(* IEC 61131-3 sources: com.logicals.lc3.webinar/logicals_Lib_Webinar/logicals_Webinar_Basic_Lib/logicals_Lib/src_FB_FBD/Logic, 6 files *)

(* ---- FB_lc_EinsAusDrei_Auswahl2_FBD.iecfbd ---- *)
NAMESPACE com.logicals.Basic.Logic
FUNCTION_BLOCK FB_lc_EinsAusDrei_Auswahl2_FBD
  {
    height := 50;
    width := 370;
  }

  VAR_INPUT
    vix_In1 : BOOL;
    vix_In2 : BOOL;
    vix_In3 : BOOL;
  END_VAR
  VAR_OUTPUT
    vox_Out : BOOL;
  END_VAR

  (*

    // Network 1:
    AND(IN1 := vix_In1, IN2 := NOT vix_In2, IN3 := NOT vix_In3, AND => @C(13).AND);
    AND(IN1 := NOT vix_In1, IN2 := vix_In2, IN3 := NOT vix_In3, AND => @C(14).AND);
    AND(IN1 := NOT vix_In1, IN2 := NOT vix_In2, IN3 := vix_In3, AND => @C(16).AND);
    OR(IN1 := @C(13).AND, IN2 := @C(14).AND, IN3 := @C(16).AND, OR => vox_Out);

  *)

  @VF(1) : @E(vix_In1), @R(560.0, 210.0, 140.0, 19.0);
  @VF(2) : @E(vix_In2), @R(560.0, 230.0, 140.0, 19.0);
  @VF(3) : @E(vix_In3), @R(560.0, 250.0, 140.0, 19.0);
  @VF(8) : @E(vox_Out), @R(1200.0, 210.0, 140.0, 19.0);
  @CF(11) : @R(30.0, 40.0, 870.0, 100.0), @T("E:$NFB_lc_EinsAusDreiAuswahl2_FBD"), @POU;
  @CF(12) : @R(1008.0, 42.6, 870.0, 100.0), @T("D:$NFB_lc_EinsAusDreiAuswahl2_FBD"), @POU;
  @C(13) : @F(AND), @R(880.0, 210.0, 40.0, 58.0), BOOL, @I(@N(IN1), @L(9.5)), @I(@N(IN2), @L(29.5), @NEG), @I(@N(IN3), @L(49.5), @NEG), @O(@N(AND), @R(9.5));
  @C(14) : @F(AND), @R(880.0, 310.0, 40.0, 58.0), BOOL, @I(@N(IN1), @L(9.5), @NEG), @I(@N(IN2), @L(29.5)), @I(@N(IN3), @L(49.5), @NEG), @O(@N(AND), @R(9.5));
  @C(15) : @F(OR), @R(1090.0, 210.0, 40.0, 58.0), BOOL, @I(@N(IN1), @L(9.5)), @I(@N(IN2), @L(29.5)), @I(@N(IN3), @L(49.5)), @O(@N(OR), @R(9.5));
  @C(16) : @F(AND), @R(880.0, 410.0, 40.0, 58.0), BOOL, @I(@N(IN1), @L(9.5), @NEG), @I(@N(IN2), @L(29.5), @NEG), @I(@N(IN3), @L(49.5)), @O(@N(AND), @R(9.5));
  @CP(4) : 731.9, 219.5;
  @CP(5) : 731.9, 317.9;
  @CP(6) : 761.0, 239.5;
  @CP(7) : 761.0, 338.2;
  @CP(9) : 790.2, 259.5;
  @CP(10) : 790.2, 354.7;

  @G(17) :
     @L(@VF(1).o, @CP(4)),
     @L(@CP(4), @C(13).IN1),
     @L(@CP(4), @CP(5)),
     @L(@CP(5), @C(14).IN1),
     @L(@CP(5), @C(16).IN1)
    ;
  @G(18) :
     @L(@VF(2).o, @CP(6)),
     @L(@CP(6), @C(13).IN2),
     @L(@CP(6), @CP(7)),
     @L(@CP(7), @C(14).IN2),
     @L(@CP(7), @C(16).IN2)
    ;
  @G(19) :
     @L(@VF(3).o, @CP(9)),
     @L(@CP(9), @C(13).IN3),
     @L(@CP(9), @CP(10)),
     @L(@CP(10), @C(14).IN3),
     @L(@CP(10), @C(16).IN3)
    ;
  @G(23) :
     @L(@C(13).AND, @C(15).IN1)
    ;
  @G(24) :
     @L(@C(14).AND, @C(15).IN2)
    ;
  @G(25) :
     @L(@C(15).OR, @VF(8).i)
    ;
  @G(27) :
     @L(@C(16).AND, @C(15).IN3)
    ;
END_FUNCTION_BLOCK
END_NAMESPACE

(* ---- FB_lc_EinsAusDrei_Auswahl3_FBD.iecfbd ---- *)
NAMESPACE com.logicals.Basic.Logic
FUNCTION_BLOCK FB_lc_EinsAusDrei_Auswahl3_FBD
  {
    width := 350;
    minWidth := 340;
    maxWidth := 340;
    height := 58;
    minHeight := 58;
    maxHeight := 58;
  }

  VAR_INPUT
    vix_In1 : BOOL;
    vix_In2 : BOOL;
    vix_In3 : BOOL;
  END_VAR
  VAR_OUTPUT
    vox_Out : BOOL;
    vox_Out1 : BOOL;
    vox_Out2 : BOOL;
    vox_Out3 : BOOL;
  END_VAR

  (*

    // Network 1:
    AND(IN1 := vix_In1, IN2 := NOT vix_In2, IN3 := NOT vix_In3, AND => @C(7).AND);
    AND(IN1 := NOT vix_In1, IN2 := vix_In2, IN3 := NOT vix_In3, AND => @C(16).AND);
    AND(IN1 := NOT vix_In1, IN2 := NOT vix_In2, IN3 := vix_In3, AND => @C(23).AND);
    OR(IN1 := @C(7).AND, IN2 := @C(16).AND, IN3 := @C(23).AND, OR => (@C(11).OR, vox_Out));
    AND(IN1 := @C(11).OR, IN2 := vix_In1, AND => vox_Out1);
    AND(IN1 := @C(11).OR, IN2 := vix_In2, AND => vox_Out2);
    AND(IN1 := @C(11).OR, IN2 := vix_In3, AND => vox_Out3);

  *)

  @CF(1) : @R(30.0, 460.0, 870.0, 100.0), @T("E:$Nlc_FB_EinsAusDreiAuswahl_FBD"), @POU;
  @CF(2) : @R(1008.0, 462.6, 870.0, 100.0), @T("D:$Nlc_FB_EinsAusDreiAuswahl_FBD"), @POU;
  @VF(3) : @E(vix_In1), @R(560.0, 630.0, 140.0, 19.0);
  @VF(4) : @E(vix_In2), @R(560.0, 650.0, 140.0, 19.0);
  @VF(5) : @E(vix_In3), @R(560.0, 670.0, 140.0, 19.0);
  @VF(6) : @E(vox_Out), @R(1370.0, 630.0, 140.0, 19.0);
  @C(7) : @F(AND), @R(880.0, 630.0, 40.0, 58.0), BOOL, @I(@N(IN1), @L(9.5)), @I(@N(IN2), @L(29.5), @NEG), @I(@N(IN3), @L(49.5), @NEG), @O(@N(AND), @R(9.5));
  @C(11) : @F(OR), @R(1090.0, 630.0, 40.0, 58.0), BOOL, @I(@N(IN1), @L(9.5)), @I(@N(IN2), @L(29.5)), @I(@N(IN3), @L(49.5)), @O(@N(OR), @R(9.5));
  @VF(13) : @E(vix_In1), @R(560.0, 730.0, 140.0, 19.0);
  @VF(14) : @E(vix_In2), @R(560.0, 750.0, 140.0, 19.0);
  @VF(15) : @E(vix_In3), @R(560.0, 770.0, 140.0, 19.0);
  @C(16) : @F(AND), @R(880.0, 730.0, 40.0, 58.0), BOOL, @I(@N(IN1), @L(9.5), @NEG), @I(@N(IN2), @L(29.5)), @I(@N(IN3), @L(49.5), @NEG), @O(@N(AND), @R(9.5));
  @VF(20) : @E(vix_In1), @R(560.0, 830.0, 140.0, 19.0);
  @VF(21) : @E(vix_In2), @R(560.0, 850.0, 140.0, 19.0);
  @VF(22) : @E(vix_In3), @R(560.0, 870.0, 140.0, 19.0);
  @C(23) : @F(AND), @R(880.0, 830.0, 40.0, 58.0), BOOL, @I(@N(IN1), @L(9.5), @NEG), @I(@N(IN2), @L(29.5), @NEG), @I(@N(IN3), @L(49.5)), @O(@N(AND), @R(9.5));
  @VF(30) : @E(vox_Out1), @R(1370.0, 730.0, 140.0, 19.0);
  @VF(31) : @E(vox_Out2), @R(1370.0, 790.0, 140.0, 19.0);
  @VF(32) : @E(vox_Out3), @R(1370.0, 850.0, 140.0, 19.0);
  @C(33) : @F(AND), @R(1290.0, 730.0, 40.0, 38.0), BOOL, @I(@N(IN1), @L(9.5)), @I(@N(IN2), @L(29.5)), @O(@N(AND), @R(9.5));
  @C(34) : @F(AND), @R(1290.0, 790.0, 40.0, 38.0), BOOL, @I(@N(IN1), @L(9.5)), @I(@N(IN2), @L(29.5)), @O(@N(AND), @R(9.5));
  @C(35) : @F(AND), @R(1290.0, 850.0, 40.0, 38.0), BOOL, @I(@N(IN1), @L(9.5)), @I(@N(IN2), @L(29.5)), @O(@N(AND), @R(9.5));
  @VF(36) : @E(vix_In1), @R(1080.0, 750.0, 140.0, 19.0);
  @VF(37) : @E(vix_In2), @R(1080.0, 810.0, 140.0, 19.0);
  @VF(38) : @E(vix_In3), @R(1080.0, 870.0, 140.0, 19.0);
  @CP(42) : 1249.5, 639.5;
  @CP(43) : 1249.5, 739.5;
  @CP(44) : 1249.5, 799.5;

  @G(8) :
     @L(@VF(3).o, @C(7).IN1)
    ;
  @G(9) :
     @L(@VF(4).o, @C(7).IN2)
    ;
  @G(10) :
     @L(@VF(5).o, @C(7).IN3)
    ;
  @G(12) :
     @L(@C(7).AND, @C(11).IN1)
    ;
  @G(17) :
     @L(@VF(13).o, @C(16).IN1)
    ;
  @G(18) :
     @L(@VF(14).o, @C(16).IN2)
    ;
  @G(19) :
     @L(@VF(15).o, @C(16).IN3)
    ;
  @G(24) :
     @L(@VF(20).o, @C(23).IN1)
    ;
  @G(25) :
     @L(@VF(21).o, @C(23).IN2)
    ;
  @G(26) :
     @L(@VF(22).o, @C(23).IN3)
    ;
  @G(27) :
     @L(@C(16).AND, @C(11).IN2)
    ;
  @G(28) :
     @L(@C(23).AND, @C(11).IN3)
    ;
  @G(29) :
     @L(@C(11).OR, @CP(42)),
     @L(@CP(42), @VF(6).i),
     @L(@CP(42), @CP(43)),
     @L(@CP(43), @C(33).IN1),
     @L(@CP(43), @CP(44)),
     @L(@CP(44), @C(34).IN1),
     @L(@CP(44), @C(35).IN1)
    ;
  @G(39) :
     @L(@VF(36).o, @C(33).IN2)
    ;
  @G(40) :
     @L(@VF(38).o, @C(35).IN2)
    ;
  @G(41) :
     @L(@VF(37).o, @C(34).IN2)
    ;
  @G(45) :
     @L(@C(33).AND, @VF(30).i)
    ;
  @G(46) :
     @L(@C(34).AND, @VF(31).i)
    ;
  @G(47) :
     @L(@C(35).AND, @VF(32).i)
    ;
END_FUNCTION_BLOCK
END_NAMESPACE

(* ---- FB_lc_ModeSelect_FBD.iecfbd ---- *)
NAMESPACE com.logicals.Basic.Logic
FUNCTION_BLOCK FB_lc_ModeSelect_FBD
  {
    height := 200;
    width := 300;
  }

  VAR
    R_TRIG1 : R_TRIG;
    lx_InitPulse : BOOL;
    Local_TRUE : BOOL;
    R_TRIG : R_TRIG;
    R_TRIG2 : R_TRIG;
    R_TRIG3 : R_TRIG;
    R_TRIG4 : R_TRIG;
    li_CycleCount : INT;
    li_Alive : INT;
    lx_CyclePulse : BOOL;
    SR1 : SR;
    SR2 : SR;
    SR3 : SR;
    SR4 : SR;
  END_VAR
  VAR_INPUT
    vix_SetHand : BOOL;
    vix_SetAutomatik : BOOL;
    vix_SetTest : BOOL;
    vix_SetSim : BOOL;
  END_VAR
  VAR_OUTPUT
    vox_Handbetrieb : BOOL;
    vox_Automatikbetrieb : BOOL;
    vox_Testbetrieb : BOOL;
    vox_Simbetrieb : BOOL;
  END_VAR

  (*

    // Network 1:
    R_TRIG(CLK := Local_TRUE, Q => lx_InitPulse);

    // Network 2:
    li_Alive := li_CycleCount;
    ADD(IN1 := li_CycleCount, IN2 := 1, ADD => li_CycleCount);

    // Network 3:
    NOT(IN := lx_CyclePulse, NOT => lx_CyclePulse);

    // Network 4:
    R_TRIG1(CLK := vix_SetHand);
    OR(IN1 := R_TRIG1.Q, IN2 := Local_TRUE, OR => @C(14).OR);
    OR(IN1 := vox_Automatikbetrieb, IN2 := vox_Testbetrieb, IN3 := vox_Simbetrieb, OR => @C(18).OR);
    SR1(S1 := @C(14).OR, R := @C(18).OR, Q1 => vox_Handbetrieb);

    // Network 5:
    R_TRIG2(CLK := vix_SetAutomatik);
    OR(IN1 := vox_Handbetrieb, IN2 := vox_Testbetrieb, IN3 := vox_Simbetrieb, OR => @C(35).OR);
    SR2(S1 := R_TRIG2.Q, R := @C(35).OR, Q1 => vox_Automatikbetrieb);

    // Network 6:
    R_TRIG3(CLK := vix_SetTest);
    OR(IN1 := vox_Handbetrieb, IN2 := vox_Automatikbetrieb, IN3 := vox_Simbetrieb, OR => @C(48).OR);
    SR3(S1 := R_TRIG3.Q, R := @C(48).OR, Q1 => vox_Testbetrieb);

    // Network 7:
    R_TRIG4(CLK := vix_SetSim);
    OR(IN1 := vox_Handbetrieb, IN2 := vox_Testbetrieb, IN3 := vox_Automatikbetrieb, OR => @C(63).OR);
    SR4(S1 := R_TRIG4.Q, R := @C(63).OR, Q1 => vox_Simbetrieb);

  *)

  @VF(1) : @E(vix_SetHand), @R(190.0, 100.0, 140.0, 19.0);
  @C(2) : @FB(R_TRIG1), @R(390.0, 100.0, 140.0, 18.5), BOOL, @I(@N(CLK), @L(9.5)), @O(@N(Q), @R(9.5));
  @VF(6) : @E(vox_Handbetrieb), @R(888.0, 99.9, 150.0, 19.0);
  @VF(8) : @E(lx_InitPulse), @R(630.0, -1180.0, 140.0, 19.0);
  @VF(9) : @E(Local_TRUE), @R(250.0, -1180.0, 140.0, 19.0);
  @C(11) : @FB(R_TRIG), @R(430.0, -1180.0, 140.0, 18.5), BOOL, @I(@N(CLK), @L(9.5)), @O(@N(Q), @R(9.5));
  @C(14) : @F(OR), @R(590.0, 100.0, 40.0, 38.0), BOOL, @I(@N(IN1), @L(9.5)), @I(@N(IN2), @L(29.5)), @O(@N(OR), @R(9.5));
  @VF(16) : @E(Local_TRUE), @R(190.0, 120.0, 140.0, 19.0);
  @C(18) : @F(OR), @R(590.0, 180.0, 40.0, 58.0), BOOL, @I(@N(IN1), @L(9.5)), @I(@N(IN2), @L(29.5)), @I(@N(IN3), @L(49.5)), @O(@N(OR), @R(9.5));
  @VF(20) : @E(vox_Automatikbetrieb), @R(190.0, 180.0, 200.0, 19.0);
  @VF(21) : @E(vox_Testbetrieb), @R(190.0, 200.0, 200.0, 19.0);
  @VF(22) : @E(vox_Simbetrieb), @R(190.0, 220.0, 200.0, 19.0);
  @VF(26) : @E(vix_SetAutomatik), @R(190.0, 300.0, 200.0, 19.0);
  @VF(28) : @E(vox_Handbetrieb), @R(190.0, 380.0, 200.0, 19.0);
  @VF(29) : @E(vox_Testbetrieb), @R(190.0, 400.0, 200.0, 19.0);
  @VF(30) : @E(vox_Simbetrieb), @R(190.0, 420.0, 200.0, 19.0);
  @VF(31) : @E(vox_Automatikbetrieb), @R(840.0, 300.0, 210.0, 19.0);
  @C(32) : @FB(R_TRIG2), @R(440.0, 300.0, 140.0, 18.5), BOOL, @I(@N(CLK), @L(9.5)), @O(@N(Q), @R(9.5));
  @C(35) : @F(OR), @R(590.0, 380.0, 40.0, 58.0), BOOL, @I(@N(IN1), @L(9.5)), @I(@N(IN2), @L(29.5)), @I(@N(IN3), @L(49.5)), @O(@N(OR), @R(9.5));
  @VF(33) : @E(vix_SetTest), @R(200.0, 520.0, 200.0, 19.0);
  @VF(37) : @E(vox_Handbetrieb), @R(200.0, 600.0, 200.0, 19.0);
  @VF(38) : @E(vox_Automatikbetrieb), @R(200.0, 620.0, 200.0, 19.0);
  @VF(41) : @E(vox_Simbetrieb), @R(200.0, 640.0, 200.0, 19.0);
  @VF(45) : @E(vox_Testbetrieb), @R(850.0, 520.0, 210.0, 19.0);
  @C(46) : @FB(R_TRIG3), @R(450.0, 520.0, 140.0, 18.5), BOOL, @I(@N(CLK), @L(9.5)), @O(@N(Q), @R(9.5));
  @C(48) : @F(OR), @R(600.0, 600.0, 40.0, 58.0), BOOL, @I(@N(IN1), @L(9.5)), @I(@N(IN2), @L(29.5)), @I(@N(IN3), @L(49.5)), @O(@N(OR), @R(9.5));
  @VF(56) : @E(vix_SetSim), @R(200.0, 740.0, 200.0, 19.0);
  @VF(57) : @E(vox_Handbetrieb), @R(200.0, 820.0, 200.0, 19.0);
  @VF(58) : @E(vox_Testbetrieb), @R(200.0, 840.0, 200.0, 19.0);
  @VF(59) : @E(vox_Automatikbetrieb), @R(200.0, 860.0, 200.0, 19.0);
  @VF(60) : @E(vox_Simbetrieb), @R(850.0, 740.0, 210.0, 19.0);
  @C(61) : @FB(R_TRIG4), @R(450.0, 740.0, 140.0, 18.5), BOOL, @I(@N(CLK), @L(9.5)), @O(@N(Q), @R(9.5));
  @C(63) : @F(OR), @R(600.0, 820.0, 40.0, 58.0), BOOL, @I(@N(IN1), @L(9.5)), @I(@N(IN2), @L(29.5)), @I(@N(IN3), @L(49.5)), @O(@N(OR), @R(9.5));
  @VF(71) : @E(li_CycleCount), @R(230.0, -890.0, 140.0, 19.0);
  @VF(72) : @E(li_CycleCount), @R(510.0, -890.0, 140.0, 19.0);
  @VF(73) : @E(1), @R(230.0, -870.0, 140.0, 19.0), INT;
  @VF(74) : @E(li_Alive), @R(760.0, -890.0, 140.0, 19.0);
  @VF(75) : @E(lx_CyclePulse), @R(290.0, -650.0, 140.0, 19.0);
  @VF(76) : @E(lx_CyclePulse), @R(640.0, -650.0, 140.0, 19.0);
  @C(79) : @F(ADD), @R(420.0, -890.0, 40.0, 38.0), INT, @I(@N(IN1), @L(9.5)), @I(@N(IN2), @L(29.5)), @I(@N(IN3), @L(49.5)), @I(@N(IN4), @L(69.5)), @I(@N(IN5), @L(89.5)), @I(@N(IN6), @L(109.5)), @I(@N(IN7), @L(129.5)), @I(@N(IN8), @L(149.5)), @I(@N(IN9), @L(169.5)), @I(@N(IN10), @L(189.5)), @I(@N(IN11), @L(209.5)), @I(@N(IN12), @L(229.5)), @I(@N(IN13), @L(249.5)), @I(@N(IN14), @L(269.5)), @I(@N(IN15), @L(289.5)), @I(@N(IN16), @L(309.5)), @O(@N(ADD), @R(9.5));
  @C(80) : @F(NOT), @R(480.0, -650.0, 60.0, 18.5), BOOL, @I(@N(IN), @L(9.5)), @O(@N(NOT), @R(9.5));
  @C(4) : @FB(SR1), @R(700.0, 100.0, 80.0, 38.0), BOOL, @I(@N(S1), @L(9.5)), @I(@N(R), @L(29.5)), @O(@N(Q1), @R(9.5));
  @C(27) : @FB(SR2), @R(700.0, 300.0, 80.0, 38.0), BOOL, @I(@N(S1), @L(9.5)), @I(@N(R), @L(29.5)), @O(@N(Q1), @R(9.5));
  @C(47) : @FB(SR3), @R(700.0, 520.0, 80.0, 38.0), BOOL, @I(@N(S1), @L(9.5)), @I(@N(R), @L(29.5)), @O(@N(Q1), @R(9.5));
  @C(62) : @FB(SR4), @R(710.0, 740.0, 80.0, 38.0), BOOL, @I(@N(S1), @L(9.5)), @I(@N(R), @L(29.5)), @O(@N(Q1), @R(9.5));
  @CF(10) : @R(430.0, -1310.0, 240.0, 100.0), @T("Lokaler InitPulse"), @POU;
  @CF(77) : @R(430.0, -1040.0, 240.0, 100.0), @T("Zyklus LifeTick"), @POU;
  @CF(78) : @R(430.0, -790.0, 240.0, 100.0), @T("Zyklus Pulse"), @POU;
  @OLT(87) : @R(70.0, 80.0, 80.0, 18.0), @S(1);
  @OLT(88) : @R(820.0, -920.0, 80.0, 18.0), @S(74);
  @OLT(89) : @R(70.0, 150.0, 80.0, 18.0), @S(20);
  @OLT(90) : @R(70.0, 180.0, 80.0, 18.0), @S(21);
  @OLT(91) : @R(70.0, 210.0, 80.0, 18.0), @S(22);
  @OLT(92) : @R(70.0, 270.0, 80.0, 18.0), @S(26);
  @OLT(93) : @R(970.0, 250.0, 80.0, 18.0), @S(31);
  @OLT(94) : @R(960.0, 60.0, 80.0, 18.0), @S(6);
  @OLT(95) : @R(980.0, 470.0, 80.0, 18.0), @S(45);

  @G(3) :
     @L(@VF(1).o, @C(2).CLK)
    ;
  @G(12) :
     @L(@C(11).Q, @VF(8).i)
    ;
  @G(13) :
     @L(@VF(9).o, @C(11).CLK)
    ;
  @G(5) :
     @L(@C(2).Q, @C(14).IN1)
    ;
  @G(17) :
     @L(@VF(16).o, @C(14).IN2)
    ;
  @G(23) :
     @L(@VF(20).o, @C(18).IN1)
    ;
  @G(24) :
     @L(@VF(21).o, @C(18).IN2)
    ;
  @G(25) :
     @L(@VF(22).o, @C(18).IN3)
    ;
  @G(36) :
     @L(@VF(26).o, @C(32).CLK)
    ;
  @G(39) :
     @L(@VF(28).o, @C(35).IN1)
    ;
  @G(40) :
     @L(@VF(29).o, @C(35).IN2)
    ;
  @G(43) :
     @L(@VF(30).o, @C(35).IN3)
    ;
  @G(49) :
     @L(@VF(33).o, @C(46).CLK)
    ;
  @G(50) :
     @L(@VF(37).o, @C(48).IN1)
    ;
  @G(51) :
     @L(@VF(38).o, @C(48).IN2)
    ;
  @G(54) :
     @L(@VF(41).o, @C(48).IN3)
    ;
  @G(64) :
     @L(@VF(56).o, @C(61).CLK)
    ;
  @G(65) :
     @L(@VF(57).o, @C(63).IN1)
    ;
  @G(66) :
     @L(@VF(58).o, @C(63).IN2)
    ;
  @G(69) :
     @L(@VF(59).o, @C(63).IN3)
    ;
  @G(81) :
     @L(@VF(71).o, @C(79).IN1)
    ;
  @G(82) :
     @L(@C(79).ADD, @VF(72).i)
    ;
  @G(83) :
     @L(@VF(73).o, @C(79).IN2)
    ;
  @G(84) :
     @L(@VF(72).o, @VF(74).i)
    ;
  @G(85) :
     @L(@VF(75).o, @C(80).IN)
    ;
  @G(86) :
     @L(@C(80).NOT, @VF(76).i)
    ;
  @G(7) :
     @L(@C(14).OR, @C(4).S1)
    ;
  @G(15) :
     @L(@C(4).Q1, @VF(6).i)
    ;
  @G(19) :
     @L(@C(18).OR, @C(4).R)
    ;
  @G(34) :
     @L(@C(32).Q, @C(27).S1)
    ;
  @G(42) :
     @L(@C(27).Q1, @VF(31).i)
    ;
  @G(44) :
     @L(@C(35).OR, @C(27).R)
    ;
  @G(52) :
     @L(@C(46).Q, @C(47).S1)
    ;
  @G(53) :
     @L(@C(47).Q1, @VF(45).i)
    ;
  @G(55) :
     @L(@C(48).OR, @C(47).R)
    ;
  @G(67) :
     @L(@C(61).Q, @C(62).S1)
    ;
  @G(68) :
     @L(@C(63).OR, @C(62).R)
    ;
  @G(70) :
     @L(@C(62).Q1, @VF(60).i)
    ;
END_FUNCTION_BLOCK
END_NAMESPACE

(* ---- FB_lc_NooM_FBD.iecfbd ---- *)
NAMESPACE com.logicals.Basic.Logic
FUNCTION_BLOCK FB_lc_NooM_FBD
  {
    vix_req2oo6 {index := 1};
    vix_req3oo6 {index := 2};
    vix_req4oo6 {index := 3};
    vix_req5oo6 {index := 4};
    vix_req6oo6 {index := 5};
    vix_a_rdy {index := 7};
    vix_b_rdy {index := 8};
    vix_c_rdy {index := 9};
    vix_d_rdy {index := 10};
    vix_e_rdy {index := 11};
    vix_f_rdy {index := 12};
    vit_sw_prio_time {index := 14};
    vit_par_time {index := 15};
    vox_req_a {index := 7};
    vox_req_b {index := 8};
    vox_req_c {index := 9};
    vox_req_d {index := 10};
    vox_req_e {index := 11};
    vox_req_f {index := 12};
  }

  VAR
    lx_reqManVisu : BOOL { description := "Manual from Visu"; };
    lxarr_Ready : ARRAY[1..16] OF BOOL;
    liarr_Prio : ARRAY[1..16] OF UINT;
    lui_NoRdy : UINT { description := "No ready"; };
    lui_NoRdyOld : UINT { description := "No ready old"; };
  END_VAR
  VAR_INPUT
    vix_req1oo6 : BOOL { description := "request 1 out of 6"; };
    vix_req2oo6 : BOOL { description := "request 2 out of 6"; };
    vix_req3oo6 : BOOL { description := "request 3 out of 6"; };
    vix_req4oo6 : BOOL { description := "request 4 out of 6"; };
    vix_req5oo6 : BOOL { description := "request 5 out of 6"; };
    vix_req6oo6 : BOOL { description := "request 6 out of 6"; };
    vix_a_rdy : BOOL { description := "a ready for operation"; };
    vix_b_rdy : BOOL { description := "b ready for operation"; };
    vix_c_rdy : BOOL { description := "c ready for operation"; };
    vix_d_rdy : BOOL { description := "d ready for operation"; };
    vix_e_rdy : BOOL { description := "e ready for operation"; };
    vix_f_rdy : BOOL { description := "f ready for operation"; };
    vit_sw_prio_time : TIME { description := "delay to change internal priorities"; };
    vit_par_time : TIME { description := "parallel operation time"; };
  END_VAR
  VAR_OUTPUT
    vox_req_a : BOOL { description := "request a"; };
    vox_req_b : BOOL { description := "request b"; };
    vox_req_c : BOOL { description := "request c"; };
    vox_req_d : BOOL { description := "request d"; };
    vox_req_e : BOOL { description := "request e"; };
    vox_req_f : BOOL { description := "request f"; };
  END_VAR

  @CF(100) : @R(370.0, 1350.0, 1158.0, 1318.0), @T("//CODE is working in CODESYS. Not testable inside this block in Logidoc. $R$N//Given here as $"additional information$"...$R$N$R$N$a0$a0$a0FOR ForCount:=1 TO 6 BY 1 DO$R$N$a0$a0$a0$a0$a0$a0IF (Ready[ForCount] = FALSE) THEN$R$N$a0$a0$a0$a0$a0$a0$a0$a0$a0Out[ForCount] := FALSE;$R$N$a0$a0$a0$a0$a0$a0END_IF;$R$N$a0$a0$a0END_FOR;$R$N$a0$a0$a0$a0$a0$R$N$a0$a0$a0Required:=0;$R$N$a0$a0$a0IF req1oo6 THEN$R$N$a0$a0$a0$a0$a0$a0Required:=1;$R$N$a0$a0$a0END_IF;$R$N$a0$a0$a0IF req2oo6 THEN $R$N$a0$a0$a0$a0$a0$a0Required:=2;$R$N$a0$a0$a0END_IF;$R$N$a0$a0$a0IF req3oo6 THEN $R$N$a0$a0$a0$a0$a0$a0Required:=3;$R$N$a0$a0$a0END_IF;$R$N$a0$a0$a0IF req4oo6 THEN $R$N$a0$a0$a0$a0$a0$a0Required:=4;$R$N$a0$a0$a0END_IF;$R$N$a0$a0$a0IF req5oo6 THEN $R$N$a0$a0$a0$a0$a0$a0Required:=5;$R$N$a0$a0$a0END_IF;$R$N$a0$a0$a0IF req6oo6 THEN $R$N$a0$a0$a0$a0$a0$a0Required :=6;$R$N$a0$a0$a0END_IF;$R$N$R$N$a0$a0$a0//internal instance of IEC-ON-Delay TON$R$N$a0$a0$a0Oscillator(IN := NOT Oscillator.Q, PT:= T#1s);$R$N$a0$a0$a0$R$N$a0$a0$a0IF Oscillator.Q = TRUE THEN$R$N$a0$a0$a0//internal ready-array$R$N$a0$a0$a0$a0$a0$a0Ready[1] := a_ready;$R$N$a0$a0$a0$a0$a0$a0Ready[2] := b_ready;$R$N$a0$a0$a0$a0$a0$a0Ready[3] := c_ready;$R$N$a0$a0$a0$a0$a0$a0Ready[4] := d_ready;$R$N$a0$a0$a0$a0$a0$a0Ready[5] := e_ready;$R$N$a0$a0$a0$a0$a0$a0Ready[6] := f_ready;$R$N$a0$a0$a0$a0$a0$a0OutCount := 0;$R$N$a0$a0$a0$a0$a0$a0ReadyCount := 0;$R$N$R$N$a0$a0$a0$a0$a0$a0$a0FOR ForCount:=1 TO 6 BY 1 DO$R$N$a0$a0$a0$a0$a0$a0$a0$a0$a0IF (Out[ForCount] = TRUE) THEN$R$N$a0$a0$a0$a0$a0$a0$a0$a0$a0$a0$a0$a0OutCount := OutCount + 1;$R$N$a0$a0$a0$a0$a0$a0$a0$a0$a0$a0$a0$a0OutOnTime[ForCount] := OutOnTime[ForCount] + 1;$R$N$a0$a0$a0$a0$a0$a0$a0$a0$a0$a0$a0$a0OutOffTime[ForCount] := 0;$R$N$a0$a0$a0$a0$a0$a0$a0$a0$a0ELSIF (Ready[ForCount] = TRUE) THEN$R$N$a0$a0$a0$a0$a0$a0$a0$a0$a0$a0$a0$a0OutOffTime[ForCount] := OutOffTime[ForCount] + 1;$R$N$a0$a0$a0$a0$a0$a0$a0$a0$a0$a0$a0$a0OutOnTime[ForCount] := 0;$R$N$a0$a0$a0$a0$a0$a0$a0$a0$a0ELSIF (Ready[ForCount] = FALSE) THEN$R$N$a0$a0$a0$a0$a0$a0$a0$a0$a0$a0$a0$a0OutOnTime[ForCount] := 0;$R$N$a0$a0$a0$a0$a0$a0$a0$a0$a0$a0$a0$a0OutOffTime[ForCount] := 0;$R$N$a0$a0$a0$a0$a0$a0$a0$a0$a0END_IF;$R$N$R$N$a0$a0$a0$a0$a0$a0$a0$a0$a0IF (Ready[ForCount] = TRUE) THEN$R$N$a0$a0$a0$a0$a0$a0$a0$a0$a0$a0$a0$a0ReadyCount := ReadyCount + 1;$R$N$a0$a0$a0$a0$a0$a0$a0$a0$a0END_IF;$R$N$a0$a0$a0$a0$a0$a0END_FOR;$R$N$R$N$R$N//CODE CONTINUES ON NEXT PAGE"), @POU;
  @CF(101) : @R(370.0, 140.0, 1148.0, 718.0), @T("inputs:$R$Na_ready = a ready for operation$R$Nb_ready = b ready for operation$R$Nc_ready = c ready for operation$R$Nd_ready = d ready for operation$R$Ne_ready = e ready for operation$R$Nf_ready = f ready for operation$R$N$R$Nreq1oo6 = 1 of the $"ready-for-operation$"-valves/drives/parts/plants a/b/c/d/e/f should start.$R$Nreq2oo6 = 2 of the $"ready-for-operation$"-valves/drives/parts/plants a/b/c/d/e/f should start.$R$Nreq3oo6 = 3 of the $"ready-for-operation$"-valves/drives/parts/plants a/b/c/d/e/f should start.$R$Nreq4oo6 = 4 of the $"ready-for-operation$"-valves/drives/parts/plants a/b/c/d/e/f should start.$R$Nreq5oo6 = 5 of the $"ready-for-operation$"-valves/drives/parts/plants a/b/c/d/e/f should start.$R$Nreq6oo6 = 6 of the $"ready-for-operation$"-valves/drives/parts/plants a/b/c/d/e/f should start.$R$N$R$Nswitch_priority_time = delay between switching priority between all $"ready-for-operation$"-valves/drives/parts/plants a/b/c/d/e/f$R$Nparallel_time = parallel operation time of requested valves/drives/parts/plants a/b/c/d/e/f when switching priority in operation$R$N$R$Noutputs:$R$Nreq_a = start valve/drive/part/plant a$R$Nreq_b = start valve/drive/part/plant b$R$Nreq_c = start valve/drive/part/plant c $R$Nreq_d = start valve/drive/part/plant d$R$Nreq_e = start valve/drive/part/plant e$R$Nreq_f = start valve/drive/part/plant f$R$N$R$N$R$Ndescription:$R$NBLOCK SELECT1 1 TO 6 OUT OF UP TO 6 valves/drives/parts/plants. $R$NBased on internal $"Runtime-ON-calculation$"/$"Runtime-OFF-calculation$" and external $"ready$"-Signal.$R$Na,b,c,d,e,f = valves/drives/parts/plants$R$N$R$N$R$N"), @POU;
  @CF(102) : @R(370.0, 2690.0, 1148.0, 1318.0), @T("//CODE CONTINUED FROM LAST PAGE$R$N$R$N$a0$a0$a0$a0$a0$a0CycleTimeCount := CycleTimeCount + 1;$R$N$a0$a0$a0$a0$a0$a0$R$N$a0$a0$a0$a0$a0$a0IF CycleTimeCount >= switch_priority_time THEN$R$N$a0$a0$a0$a0$a0$a0$a0$a0$a0CycleTimeCount := 0;$R$N$a0$a0$a0$a0$a0$a0$a0$a0$a0parallelFlag := TRUE;$R$N$a0$a0$a0$a0$a0$a0END_IF;$R$N$R$N$a0$a0$a0$a0$a0$a0IF ((parallelFlag = TRUE) AND (NOT req6oo6)) THEN$R$N$a0$a0$a0$a0$a0$a0$a0$a0$a0parallelTimeCount := parallelTimeCount + 1;$R$N$a0$a0$a0$a0$a0$a0$a0$a0$a0RequiredExt := Required + 1;$R$N$a0$a0$a0$a0$a0$a0ELSE$R$N$a0$a0$a0$a0$a0$a0$a0$a0$a0RequiredExt := Required;$R$N$a0$a0$a0$a0$a0$a0END_IF;$R$N$R$N$a0$a0$a0$a0$a0$a0IF (parallelTimeCount >= parallel_time) THEN$R$N$a0$a0$a0$a0$a0$a0$a0$a0$a0parallelTimeCount := 0;$R$N$a0$a0$a0$a0$a0$a0$a0$a0$a0parallelFlag := FALSE;$R$N$a0$a0$a0$a0$a0$a0END_IF;$R$N$R$N$a0$a0$a0$a0$a0$a0IF (ReadyCount > RequiredExt) THEN$R$N$a0$a0$a0$a0$a0$a0$a0$a0$a0WHILE (OutCount < RequiredExt) DO$R$N$a0$a0$a0$a0$a0$a0$a0$a0$a0$a0$a0$a0OldValueTime := 0;$R$N$a0$a0$a0$a0$a0$a0$a0$a0$a0$a0$a0$a0SearchRes := 1;$R$N$a0$a0$a0$a0$a0$a0$a0$a0$a0$a0$a0$a0FOR ForCount:=1 TO 6 BY 1 DO$R$N$a0$a0$a0$a0$a0$a0$a0$a0$a0$a0$a0$a0$a0$a0$a0IF ((OutOffTime[ForCount] > OldValueTime) AND (Ready[ForCount] = TRUE) AND (Out[ForCount] = FALSE)) THEN$R$N$a0$a0$a0$a0$a0$a0$a0$a0$a0$a0$a0$a0$a0$a0$a0$a0$a0$a0OldValueTime := OutOffTime[ForCount];$R$N$a0$a0$a0$a0$a0$a0$a0$a0$a0$a0$a0$a0$a0$a0$a0$a0$a0$a0SearchRes := ForCount;$R$N$a0$a0$a0$a0$a0$a0$a0$a0$a0$a0$a0$a0$a0$a0$a0END_IF;$R$N$a0$a0$a0$a0$a0$a0$a0$a0$a0$a0$a0$a0END_FOR;$R$N$a0$a0$a0$a0$a0$a0$a0$a0$a0$a0$a0$a0IF (Ready[SearchRes] = TRUE) THEN$R$N$a0$a0$a0$a0$a0$a0$a0$a0$a0$a0$a0$a0$a0$a0$a0Out[SearchRes] := TRUE;$R$N$a0$a0$a0$a0$a0$a0$a0$a0$a0$a0$a0$a0$a0$a0$a0OutCount := OutCount + 1;$R$N$a0$a0$a0$a0$a0$a0$a0$a0$a0$a0$a0$a0END_IF;$R$N$a0$a0$a0$a0$a0$a0$a0$a0$a0END_WHILE;$R$N$a0$a0$a0$a0$a0$a0ELSE$R$N$a0$a0$a0$a0$a0$a0$a0$a0$a0FOR ForCount:=1 TO 6 BY 1 DO$R$N$a0$a0$a0$a0$a0$a0$a0$a0$a0$a0$a0$a0IF (Ready[ForCount] = TRUE) THEN$R$N$a0$a0$a0$a0$a0$a0$a0$a0$a0$a0$a0$a0$a0$a0$a0Out[ForCount] := TRUE;$R$N$a0$a0$a0$a0$a0$a0$a0$a0$a0$a0$a0$a0END_IF;$R$N$a0$a0$a0$a0$a0$a0$a0$a0$a0END_FOR;$R$N$a0$a0$a0$a0$a0$a0END_IF;$R$N$R$N$a0$a0$a0$a0$a0$a0WHILE (OutCount > RequiredExt) DO$R$N$a0$a0$a0$a0$a0$a0$a0$a0$a0OldValueTime := 0;$R$N$a0$a0$a0$a0$a0$a0$a0$a0$a0SearchRes := 1;$R$N$a0$a0$a0$a0$a0$a0$a0$a0$a0FOR ForCount:=1 TO 6 BY 1 DO$R$N$a0$a0$a0$a0$a0$a0$a0$a0$a0$a0$a0$a0IF ((OutOnTime[ForCount] > OldValueTime) AND (Ready[ForCount] = TRUE) AND (Out[ForCount] = TRUE)) THEN$R$N$a0$a0$a0$a0$a0$a0$a0$a0$a0$a0$a0$a0$a0$a0$a0OldValueTime := OutOnTime[ForCount];$R$N$a0$a0$a0$a0$a0$a0$a0$a0$a0$a0$a0$a0$a0$a0$a0SearchRes := ForCount;$R$N$a0$a0$a0$a0$a0$a0$a0$a0$a0$a0$a0$a0END_IF;$R$N$a0$a0$a0$a0$a0$a0$a0$a0$a0END_FOR;$R$N$a0$a0$a0$a0$a0$a0$a0$a0$a0Out[SearchRes] := FALSE;$R$N$a0$a0$a0$a0$a0$a0$a0$a0$a0OutCount := OutCount - 1;$R$N$a0$a0$a0$a0$a0$a0END_WHILE;$R$N$a0$a0$a0END_IF;$R$N$a0$a0$a0req_a := Out[1];$R$N$a0$a0$a0req_b := Out[2];$R$N$a0$a0$a0req_c := Out[3];$R$N$a0$a0$a0req_d := Out[4];$R$N$a0$a0$a0req_e := Out[5];$R$N$a0$a0$a0req_f := Out[6];"), @POU;

  @PAGE(103) : @R(0.0, 0.0, 1900.0, 1340.0), @LN("select n out of m ");
  @PAGE(104) : @R(0.0, 1340.0, 1900.0, 1340.0), @LN("example-Code for CODESYS");
END_FUNCTION_BLOCK
END_NAMESPACE

(* ---- FB_lc_Toggle1_FBD.iecfbd ---- *)
NAMESPACE com.logicals.Basic.Logic
FUNCTION_BLOCK FB_lc_Toggle1_FBD
  VAR
    R_TRIG1 : R_TRIG;
  END_VAR
  VAR_INPUT
    vix_In : BOOL;
  END_VAR
  VAR_OUTPUT
    vox_Out : BOOL;
  END_VAR

  (*

    // Network 1:
    R_TRIG1(CLK := vix_In);
    XOR(IN1 := R_TRIG1.Q, IN2 := vox_Out, XOR => vox_Out);

  *)

  @VF(1) : @E(vix_In), @R(170.0, 100.0, 140.0, 19.0);
  @VF(2) : @E(vox_Out), @R(720.0, 100.0, 140.0, 19.0);
  @C(3) : @FB(R_TRIG1), @R(360.0, 100.0, 140.0, 18.5), @I(@N(CLK), @L(9.5)), @O(@N(Q), @R(9.5));
  @C(5) : @F(XOR), @R(580.0, 100.0, 50.0, 38.0), BOOL, @I(@N(IN1), @L(9.5)), @I(@N(IN2), @L(29.5)), @O(@N(XOR), @R(9.5));
  @VF(8) : @E(vox_Out), @R(360.0, 120.0, 140.0, 19.0);
  @CF(10) : @R(170.0, 30.0, 690.0, 50.0), @T("Toggle 1"), @POU;

  @G(4) :
     @L(@VF(1).o, @C(3).CLK)
    ;
  @G(6) :
     @L(@C(3).Q, @C(5).IN1)
    ;
  @G(7) :
     @L(@C(5).XOR, @VF(2).i)
    ;
  @G(9) :
     @L(@VF(8).o, @C(5).IN2)
    ;
END_FUNCTION_BLOCK
END_NAMESPACE

(* ---- FB_lc_ToggleSw_FBD.iecfbd ---- *)
NAMESPACE com.logicals.Basic.Logic
FUNCTION_BLOCK FB_lc_ToggleSw_FBD
  VAR
    R_TRIG : R_TRIG;
    RS : RS;
  END_VAR
  VAR_INPUT
    vix_Set : BOOL;
    vix_Trg : BOOL;
    vix_Reset : BOOL;
  END_VAR
  VAR_OUTPUT
    vox_Out : BOOL;
  END_VAR

  (*

    // Network 1:
    R_TRIG(CLK := vix_Trg);
    AND(IN1 := NOT vox_Out, IN2 := R_TRIG.Q, AND => @C(117).AND);
    OR(IN1 := vix_Set, IN2 := @C(117).AND, OR => @C(113).OR);
    AND(IN1 := R_TRIG.Q, IN2 := vox_Out, AND => @C(116).AND);
    OR(IN1 := @C(116).AND, IN2 := vix_Reset, OR => @C(114).OR);
    RS(S := @C(113).OR, R1 := @C(114).OR, Q1 => vox_Out);

  *)

  @C(115) : @FB(R_TRIG), @R(680.0, 660.0, 140.0, 18.0), @I(@N(CLK), @L(9.5)), @O(@N(Q), @R(9.5));
  @C(111) : @FB(RS), @R(1060.0, 640.0, 80.0, 38.0), @I(@N(S), @L(9.5)), @I(@N(R1), @L(29.5)), @O(@N(Q1), @R(9.5));
  @C(116) : @F(AND), @R(890.0, 660.0, 40.0, 38.0), BOOL, @I(@N(IN1), @L(9.5)), @I(@N(IN2), @L(29.5)), @O(@N(AND), @R(9.5));
  @C(114) : @F(OR), @R(980.0, 660.0, 40.0, 38.0), BOOL, @I(@N(IN1), @L(9.5)), @I(@N(IN2), @L(29.5)), @O(@N(OR), @R(9.5));
  @C(117) : @F(AND), @R(890.0, 620.0, 40.0, 38.0), BOOL, @I(@N(IN1), @L(9.5), @NEG), @I(@N(IN2), @L(29.5)), @O(@N(AND), @R(9.5));
  @C(113) : @F(OR), @R(980.0, 600.0, 40.0, 38.0), BOOL, @I(@N(IN1), @L(9.5)), @I(@N(IN2), @L(29.5)), @O(@N(OR), @R(9.5));
  @VF(105) : @E(vox_Out), @R(1800.0, 640.0, 100.0, 19.0);
  @VF(112) : @E(vox_Out), @R(680.0, 620.0, 140.0, 19.0);
  @VF(101) : @E(vix_Set), @R(0.0, 600.0, 100.0, 19.0);
  @VF(109) : @E(vix_Trg), @R(0.0, 660.0, 100.0, 19.0);
  @VF(107) : @E(vix_Reset), @R(0.0, 720.0, 100.0, 19.0);
  @CF(100) : @R(130.0, 620.0, 298.0, 18.0), @T("%l"), @S(101);
  @CF(108) : @R(130.0, 680.0, 298.0, 18.0), @T("%l"), @S(109);
  @CF(106) : @R(130.0, 740.0, 298.0, 18.0), @T("%l"), @S(107);
  @CF(102) : @R(190.0, 80.0, 728.0, 228.0), @T("E:$R$N$R$NToggle Flipflop Switch$R$N$R$NTrg-input: at 0/1-edge toggle flipflop state$R$NRes-input: at 1-signal reset flipflop (priority)$R$NSet-input: at 1-signal set flipflop$R$N$R$NY-output: $a0actual toggle flipflop state"), @POU;
  @CF(103) : @R(980.0, 80.0, 728.0, 228.0), @T("D:$R$N$R$NToggle Flipflop Schalter$R$N$R$NTrg-Eing.: bei 0/1-Flanke Flipflop umschalten$R$NRes-Eing.: bei 1-Signal Flipflop r$fccksetzen (Priorit$e4t)$R$NSet-Eing.: bei 1-Signal Flipflop setzen$R$N$R$NY-Ausgang: aktueller Toggle Flipflop Zustand"), @POU;
  @CP(127) : 870.0, 669.5;
  @CP(129) : 850.0, 629.5;

  @G(123) :
     @L(@VF(107).o, @C(114).IN2)
    ;
  @G(122) :
     @L(@C(116).AND, @C(114).IN1)
    ;
  @G(126) :
     @L(@C(115).Q, @CP(127)),
     @L(@CP(127), @C(116).IN1),
     @L(@CP(127), @C(117).IN2)
    ;
  @G(132) :
     @L(@C(114).OR, @C(111).R1)
    ;
  @G(119) :
     @L(@C(111).Q1, @VF(105).i)
    ;
  @G(130) :
     @L(@C(113).OR, @C(111).S)
    ;
  @G(121) :
     @L(@C(117).AND, @C(113).IN2)
    ;
  @G(128) :
     @L(@VF(112).o, @CP(129)),
     @L(@CP(129), @C(116).IN2),
     @L(@CP(129), @C(117).IN1)
    ;
  @G(120) :
     @L(@VF(101).o, @C(113).IN1)
    ;
  @G(125) :
     @L(@VF(109).o, @C(115).CLK)
    ;
END_FUNCTION_BLOCK
END_NAMESPACE
